Fanuc KAREL source: kt00254.KL

PROGRAM KT00254
%STACKSIZE=65535
%PRIORITY=65535
%NOLOCKGROUP
VAR
H1 : ARRAY[2] OF SHORT
Y2 : ARRAY[2] OF BYTE
OUT : INTEGER
BEGIN
H1[1]=2
Y2[1]=3
-- UNRESOLVED_PC line 10 opcodes [22 9D 33 B3 22 9D 33 B1 47 23] marker_code=38
END KT00254
